# EPICS StreamDevice protocol: protocols/qen.proto
Terminator = LF;
ExtraInput = Ignore;

clr_qen_count {
	out "qen_count 0";
	in;
}

di4_mon {
	out "di4_mon";
	in "%x";
}

read_qen_count {
	out "qen_count";
	in "%d";
}

read_z_count {
	out "zcount";
	in "%d";
}
read_e_count {
	out "ecount";
	in "%d";
}

get_tr {
	out "\$1";
	in "%d";
}

set_tr {
	out "\$1 %d";
	in;
}

set_tr3 {
        out "\$1_en 0";
        in;
        out "\$1_count %d";
        in;
        out "\$1_en 1";
        in;
}

get_en {
	out "\$1";
	in "%d";
}

set_en {
	out "\$1 %d";
	in;
}
